(* IEC 61131-3 sources: eCockpitGit/test_project/src/%F%00 Library/%F%Common Functions/%F%String/%F%Big Input/%F%Padd, 4 files *)

(* ---- %POU%FU_sPaddBackBI.st ---- *)
//This function padds the back of a string with the given character, the given amount
//If the padd amount plus the string is longer than the output string, the input string will be cut off to make space for the padding
// +-----------+----------+----------+-----------------------------------------------------------------------------------------------------------------------+
// |**Version**|**Author**| **Date** |**Changes**                                                                                                            |
// +-----------+----------+----------+-----------------------------------------------------------------------------------------------------------------------+
// | 1         | NSN      | 04-02-19 | Creation                                                                                                              |
// +-----------+----------+----------+-----------------------------------------------------------------------------------------------------------------------+
FUNCTION FU_sPaddBackBI : STRING(255)
VAR_IN_OUT
	sStr		:STRING(1);			//Input String
END_VAR
VAR_INPUT
	wPadds		:WORD;				//How much to padd it
	eChar		:EASCII;		//Which character to padd with
END_VAR
(*%!%__DELIMITER__%!%*)
FU_sPaddBackBIBO(sOut:=FU_sPaddBackBI,sStr:=sStr,wPadds:=wPadds,wOutSize:=255,eChar:=eChar);

(* ---- %POU%FU_sPaddBackLenBI.st ---- *)
//This function padds the back of a string with the given character, the given amount
//If the padd amount plus the string is longer than the output string, the input string will be cut off to make space for the padding
// +-----------+----------+----------+-----------------------------------------------------------------------------------------------------------------------+
// |**Version**|**Author**| **Date** |**Changes**                                                                                                            |
// +-----------+----------+----------+-----------------------------------------------------------------------------------------------------------------------+
// | 1         | NSN      | 04-02-19 | Creation                                                                                                              |
// +-----------+----------+----------+-----------------------------------------------------------------------------------------------------------------------+
FUNCTION FU_sPaddBackLenBI  : STRING(255)
VAR_IN_OUT
	sStr		:STRING(1);			//Input String
END_VAR
VAR_INPUT
	wLen		:WORD;				//How much to padd it
	eChar		:EASCII;		//Which character to padd with
END_VAR
(*%!%__DELIMITER__%!%*)
FU_sPaddBackLenBIBO(sOut:=FU_sPaddBackLenBI,sStr:=sStr,wLen:=wLen,wOutSize:=255,eChar:=eChar);

(* ---- %POU%FU_sPaddFrontBI.st ---- *)
//This function padds the front of a string with the given character, the given amount
//If the padd amount plus the string is longer than the output string, the input string will be cut off to make space for the padding
// +-----------+----------+----------+-----------------------------------------------------------------------------------------------------------------------+
// |**Version**|**Author**| **Date** |**Changes**                                                                                                            |
// +-----------+----------+----------+-----------------------------------------------------------------------------------------------------------------------+
// | 1         | NSN      | 04-02-19 | Creation                                                                                                              |
// +-----------+----------+----------+-----------------------------------------------------------------------------------------------------------------------+
FUNCTION FU_sPaddFrontBI : STRING(255)
VAR_IN_OUT
	sStr		:STRING(1);			//Input String
END_VAR
VAR_INPUT
	wPadds		:WORD;				//How much to padd it
	eChar		:EASCII;		//Which character to padd with
END_VAR
(*%!%__DELIMITER__%!%*)
FU_sPaddFrontBIBO(sOut:=FU_sPaddFrontBI,sStr:=sStr,wPadds:=wPadds,wOutSize:=255,eChar:=eChar);

(* ---- %POU%FU_sPaddFrontLenBI.st ---- *)
//This function padds the front of a string with the given character, the given amount
//If the padd amount plus the string is longer than the output string, the input string will be cut off to make space for the padding
// +-----------+----------+----------+-----------------------------------------------------------------------------------------------------------------------+
// |**Version**|**Author**| **Date** |**Changes**                                                                                                            |
// +-----------+----------+----------+-----------------------------------------------------------------------------------------------------------------------+
// | 1         | NSN      | 04-02-19 | Creation                                                                                                              |
// +-----------+----------+----------+-----------------------------------------------------------------------------------------------------------------------+
FUNCTION FU_sPaddFrontLenBI : STRING(255)
VAR_IN_OUT
	sStr		:STRING(1);			//Input String
END_VAR
VAR_INPUT
	wLen		:WORD;				//How much to padd it
	eChar		:EASCII;		//Which character to padd with
END_VAR
(*%!%__DELIMITER__%!%*)
FU_sPaddFrontLenBIBO(sOut:=FU_sPaddFrontLenBI,sStr:=sStr,wLen:=wLen,wOutSize:=255,eChar:=eChar);
